(* IEC 61131-3 sources: axopen.templates/axopen.template.simple/ax/src/templates/unit, 7 files *)

(* ---- AutomatSequence.st ---- *)
NAMESPACE axosimple.UnitTemplate
    USING axosimple;
    USING AXOpen.Data;
    USING AXOpen.Core;
    USING System.Strings;

    ///<summary>
    /// Provides automatic mode sequence.
    ///</summary>
    {#ix-set:AttributeName = "<#AUTOMAT#>"}
    {S7.extern=ReadWrite}
    CLASS PUBLIC AutomatSequence
        EXTENDS AXOpen.Core.AxoSequencerContainer
        IMPLEMENTS IModeContainer
        VAR PUBLIC
            Steps : ARRAY[0..150] OF AXOpen.Core.AxoStep;
        END_VAR
        VAR PRIVATE
            Objs : axosimple.UnitTemplate.UnitObjects;
            _currentId : STRING;
        END_VAR

        METHOD INTERNAL Run
            VAR_INPUT
                inParent :  AXOpen.Core.IAxoObject;
                inUnitObjects : REF_TO axosimple.UnitTemplate.UnitObjects;
            END_VAR

            SUPER.Run(inParent);
        END_METHOD
        ///<summary>
        /// Contains logic of the steps of this sequence
        ///</summary>

        METHOD OVERRIDE Main
            // This sequecner executes the steps in cycles from top to bottom
            // in the same order they are written in the program
            // Each step in the sequence must can be used only once.
            // This sets the sequence to run in cycles (top-botton-top and again).
            THIS.SequenceMode := eAxoSequenceMode#Cyclic;

            IF (Steps[0].Execute(THIS, TRUE, '<#GET ID#>')) THEN
                //-------------------------------------------------------
                _currentId := 'newProducedPart';
                THIS.MoveNext();
                //-------------------------------------------------------
            END_IF;

            IF (Steps[10].Execute(THIS, TRUE, '<#GET DATA#>')) THEN
                //-------------------------------------------------------
                // IF(ProcessSettingsManager^.Read('MODEL_S').IsDone()) THEN
                //     ProcessDataManager^.DataManger.Payload := ProcessSettingsManager^.Payload;
                //     THIS.MoveNext();
                // END_IF;

                RETURN;

                IF (Objs.ProcessData.CreateOrUpdate(_currentId).IsDone()) THEN
                    THIS.MoveNext();
                END_IF;

                //-------------------------------------------------------
            END_IF;

            IF (Steps[20].Execute(THIS, TRUE, '<#DO SOMETHING#>')) THEN
                //-------------------------------------------------------

                IF(Objs.ProcessData.DataManger.Payload.JigDataMatrixCode.Inspect(THIS, '').Done()) THEN
                    THIS.MoveNext();
                END_IF;
                //-------------------------------------------------------
            END_IF;

            IF (Steps[30].Execute(THIS, TRUE, '<#DO SOMETHING#>')) THEN
                //-------------------------------------------------------
                IF(Objs.ProcessData.DataManger.Payload.PartPresence.Inspect(THIS, TRUE).Done()) THEN
                    THIS.MoveNext();
                END_IF;
                //-------------------------------------------------------
            END_IF;

            IF (Steps[4].Execute(THIS, TRUE, '<#DO SOMETHING#>')) THEN
                //-------------------------------------------------------
                IF(Objs.ProcessData.DataManger.Payload.RivetingPreasure.Inspect(THIS, 1.5).Done()) THEN
                    THIS.MoveNext();
                END_IF;
                //-------------------------------------------------------
            END_IF;

            IF (Steps[149].Execute(THIS, TRUE, '<#UPDATE DATA#>')) THEN
                //-------------------------------------------------------
                IF (Objs.ProcessData.Update(_currentId).IsDone()) THEN
                    THIS.MoveNext();
                END_IF;
                //-------------------------------------------------------
            END_IF;

            // This will close the sequence and will return to the first step.
            THIS.Close(Steps[150]);
        END_METHOD
    END_CLASS
END_NAMESPACE

(* ---- Components.st ---- *)
NAMESPACE axosimple.UnitTemplate
    USING axosimple;
    USING AXOpen.Data;
    USING AXOpen.Core;
    USING System.Strings;

    ///<summary>
    /// Groups components of this controller unit.
    ///</summary>
    {S7.extern=ReadWrite}
    CLASS Components
        EXTENDS AXOpen.Core.AxoObject
        VAR PUBLIC
            // HERE DECLARE COMPONENTS USED BY THIS CONTROLLED UNIT
            HorizontalCylinder : AXOpen.Components.Pneumatics.AxoCylinder;
            VerticalCylinder : AXOpen.Components.Pneumatics.AxoCylinder;
            GripperCylinder : AXOpen.Components.Pneumatics.AxoCylinder;
        END_VAR

        METHOD PUBLIC Update
            VAR_INPUT
                parent : IAxoObject;
                Inputs : ref_to axosimple.Inputs; // must be a ref_to due to arrays in components
                Outputs : ref_to axosimple.Outputs;
            END_VAR
            THIS.Initialize(parent);

            THIS.Initialize(parent);
            // HERE INITIALIZE YOUR COMPONENTS
            HorizontalCylinder.Run(THIS, Inputs^.P0[0], Inputs^.P0[1], Outputs^.P0[0], Outputs^.P0[1]);
            VerticalCylinder.Run(THIS, Inputs^.P0[2], Inputs^.P0[3], Outputs^.P0[2], Outputs^.P0[3]);
            GripperCylinder.Run(THIS, Inputs^.P0[4], Inputs^.P0[5], Outputs^.P0[4], Outputs^.P0[5]);

        END_METHOD
    END_CLASS
END_NAMESPACE

(* ---- GroundSequence.st ---- *)
NAMESPACE axosimple.UnitTemplate
    USING axosimple;
    USING AXOpen.Data;
    USING AXOpen.Core;
    USING System.Strings;

    ///<summary>
    /// Provides ground mode sequence.
    ///</summary>
    {#ix-set:AttributeName = "<#GROUND#>"}
    {S7.extern=ReadWrite}
    CLASS PUBLIC GroundSequence
        EXTENDS AXOpen.Core.AxoSequencerContainer
        IMPLEMENTS IModeContainer
        VAR PUBLIC
            Steps : ARRAY[0..20] OF AXOpen.Core.AxoStep;
            MoveToWork : AXOpen.Core.AxoTask;
        END_VAR
        VAR PRIVATE
            Objs : REF_TO axosimple.UnitTemplate.UnitObjects;
            Components : REF_TO axosimple.UnitTemplate.Components;

            ProcessDataManager : REF_TO axosimple.UnitTemplate.ProcessDataManager;
            ProcessSettingsManager : REF_TO axosimple.UnitTemplate.FragmentProcessDataManger;
            TechnologySettingsManager : REF_TO axosimple.UnitTemplate.TechnologyDataManager;

            PersistentSettingsManager : REF_TO AxoDataPersistentExchange;

            _currentId : STRING;

            techSetttingsId : STRING;
        END_VAR

        METHOD INTERNAL Run
            VAR_INPUT
                inParent : AXOpen.Core.IAxoObject;
                inUnitObjects : REF_TO axosimple.UnitTemplate.UnitObjects;
            END_VAR

            IF Objs = NULL THEN
                Objs := inUnitObjects;
            END_IF;

            SUPER.Run(inParent);

        END_METHOD
        ///<summary>
        /// Contains logic of the steps of this sequence
        ///</summary>

        METHOD PROTECTED OVERRIDE Main
            // IF (Components = NULL OR ProcessData = NULL) THEN
            //     RETURN;
            // END_IF;
            // This sequecner executes the steps in cycles from top to bottom
            // in the same order they are written in the program
            // Each step in the sequence must can be used only once.
            // This sets the sequence to run once (top-botton) and stops with done after closing.
            THIS.SequenceMode := eAxoSequenceMode#RunOnce;

            IF (Steps[0].Execute(THIS, TRUE, '<#RESTORE#>')) THEN
                //-------------------------------------------------------
                    TechnologySettingsManager^.Restore();
                    ProcessSettingsManager^.Restore();
                    ProcessDataManager^.Restore();

                    THIS.MoveNext();
                //-------------------------------------------------------
            END_IF;

            IF (Steps[1].Execute(THIS, TRUE, '<#READ PERSISTENT SETTINGS#>')) THEN
                //-------------------------------------------------------
                CASE TO_INT( THIS.GetMicroStepValue()) OF
                    0 :
                        IF PersistentSettingsManager^.InvokeRead(THIS,'UnitTemplate') THEN
                            THIS.SetMicroStepValue(UINT#10);
                        END_IF;
                    10 :
                        IF PersistentSettingsManager^.IsReadDone(THIS) THEN
                                THIS.MoveNext();
                        END_IF;
                    ELSE
                        THIS.SetMicroStepValue(UINT#0);
                END_CASE;
                //-------------------------------------------------------
            END_IF;

            IF (Steps[5].Execute(THIS, TRUE, '<#READ TECHNOLOGY SETTINS#>')) THEN
                //-------------------------------------------------------
                IF CurrentStep.IsFirstEntryToStep() THEN

                    IF Objs^.Global^.TechnologySettings^.Common.Entity.DataEntityId <> '' THEN
                       techSetttingsId := Objs^.Global^.TechnologySettings^.Common.Entity.DataEntityId; // TAKE GLOGAL TECHNOLOGY SETTINGS ID

                    ELSIF Objs^.TechnologySettings^.Payload.DataEntityId <> '' THEN // TAKE LAST LOADED FOR STATION
                        techSetttingsId := Objs^.TechnologySettings^.Payload.DataEntityId;

                    ELSIF Objs^.LastTechnologySettings <> '' THEN // TAKE LAST LOADED FROM PERSISTENT
                        techSetttingsId := Objs^.LastTechnologySettings;
                    ELSE
                        Objs^.LastTechnologySettings := 'default'; // FORCE DEFAULT VALUE
                        techSetttingsId := Objs^.LastTechnologySettings;
                    END_IF;

                    IF Objs^.Global^.TechnologySettings^.Common.Entity.DataEntityId = Objs^.TechnologySettings^.Payload.DataEntityId then
                        //THIS.MoveNext(); // you can skip loading...
                        ;
                    end_if;

                else
                    IF(TechnologySettingsManager^.Read( techSetttingsId ).IsDone()) THEN
                        THIS.MoveNext();
                    END_IF;
                END_IF;
                //-------------------------------------------------------
            END_IF;

            IF (Steps[3].Execute(THIS, TRUE, '<#DO SOMETHING#>')) THEN
                //-------------------------------------------------------
                IF CurrentStep.Duration > TIME#2s THEN
                    THIS.MoveNext();
                END_IF;
                //-------------------------------------------------------
            END_IF;

            IF (Steps[19].Execute(THIS, TRUE, '<#SAVE DATA#>')) THEN
                //-------------------------------------------------------
                CASE TO_INT( THIS.GetMicroStepValue()) OF
                    0 :
                        IF ProcessDataManager^.Shared.Entity.DataEntityId <> '' THEN
                            _currentId := ProcessDataManager^.Shared.Entity.DataEntityId;
                            THIS.SetMicroStepValue(UINT#10);

                        ELSE // FIST RUN OR WITHOUT DATA
                            THIS.MoveNext();
                        END_IF;

                    10 : // update part as a corrupted a interrupted
                        ProcessDataManager^.Shared.Entity.WasReset := true;
                        IF ProcessDataManager^.Update(_currentId).IsDone() THEN
                                THIS.MoveNext();
                        END_IF;
                    ELSE
                        THIS.SetMicroStepValue(UINT#0);
                END_CASE;
                //-------------------------------------------------------
            END_IF;

            // This will close the sequence and will return to the first step.
            THIS.Close(Steps[20]);
        END_METHOD
    END_CLASS
END_NAMESPACE

(* ---- ProcessData.st ---- *)
NAMESPACE axosimple.UnitTemplate
    USING axosimple;
    USING AXOpen.Data;
    USING AXOpen.Core;
    USING System.Strings;

    {S7.extern=ReadWrite}
    CLASS ProcessData
        EXTENDS AXOpen.Data.AxoDataEntity
        VAR PUBLIC
            Header : axosimple.UnitHeader;
            DimX    : AXOpen.Inspectors.AxoAnalogueInspector;
            DimY    : AXOpen.Inspectors.AxoAnalogueInspector;
            DimZ    : AXOpen.Inspectors.AxoAnalogueInspector;
        END_VAR
    END_CLASS
END_NAMESPACE

(* ---- ServiceMode.st ---- *)
NAMESPACE axosimple.UnitTemplate
    USING axosimple;
    USING AXOpen.Data;
    USING AXOpen.Core;
    USING System.Strings;

    ///<summary>
    /// Provides logic for service/manual/maintenance mode.
    ///</summary>
    {#ix-set:AttributeName = "<#SERVICE#>"}
    {S7.extern=ReadWrite}
    CLASS PUBLIC ServiceMode
        EXTENDS AXOpen.Core.AxoTask
        IMPLEMENTS IModeContainer
        ///<summary>
        /// Runs service mode logic. This method must be called cyclically.
        ///</summary>

        METHOD PUBLIC Run
            VAR_INPUT
                parent : AXOpen.Core.IAxoObject;
            END_VAR
            VAR_IN_OUT
                components : axosimple.UnitTemplate.Components;
            END_VAR
            THIS.Initialize(parent);
            IF THIS.Execute() THEN
                THIS.Handle(components);
            END_IF;
        END_METHOD

        METHOD PRIVATE Handle
            VAR_IN_OUT
                components : axosimple.UnitTemplate.Components;
            END_VAR
            ;
            // HERE CALL LOGIC FOR MANUAL/SERICE OPERATIONS

            components.DI_1.ActivateManualControl();
            components.DI_2.ActivateManualControl();
            // components.DI_3.ActivateManualControl();
            // components.DI_4.ActivateManualControl();

            components.DO_1.ActivateManualControl();
            components.DO_2.ActivateManualControl();
            // components.DO_3.ActivateManualControl();
            // components.DO_4.ActivateManualControl();

            components.AI_1.ActivateManualControl();
            components.AI_2.ActivateManualControl();
            // components.AI_3.ActivateManualControl();
            // components.AI_4.ActivateManualControl();

            components.AO_1.ActivateManualControl();
            components.AO_2.ActivateManualControl();
            // components.AO_3.ActivateManualControl();
            // components.AO_4.ActivateManualControl();

            components.Cylinder_1.ActivateManualControl();
            components.Cylinder_2.ActivateManualControl();
            // components.Cylinder_3.ActivateManualControl();
            // components.Cylinder_4.ActivateManualControl();

            // components.Reader_1.ActivateManualControl();
            // components.Reader_2.ActivateManualControl();

            // components.Camera_1.ActivateManualControl();
            // components.Camera_2.ActivateManualControl();

            // components.Drive_R1.ActivateManualControl();
            // components.Drive_R2.ActivateManualControl();

            // components.Drive_F1.ActivateManualControl();
            // components.Drive_F2.ActivateManualControl();

        END_METHOD
    END_CLASS
END_NAMESPACE

(* ---- Unit.st ---- *)
NAMESPACE axosimple.UnitTemplate
    USING axosimple;
    USING AXOpen.Data;
    USING AXOpen.Core;
    USING System.Strings;

    ///<summary>
    /// Represents controlled units and high level task coordination.
    ///</summary>
    {S7.extern=ReadWrite}
    CLASS Unit
        EXTENDS axosimple.BaseUnit.UnitBase
        VAR PUBLIC
            ///<summary>
            /// Provide access to unit objets, that are used into sequnces.
            ///</summary>
            UnitObjects  : axosimple.UnitTemplate.UnitObjects;

            ///<summary>
            /// Ground sequence. Contains logic that brings the unit into initial state.
            ///</summary>
            GroundSequence : axosimple.UnitTemplate.GroundSequence;

            ///<summary>
            /// Automatic sequence. Contains logic for automatic operations of this unit.
            ///</summary>
            AutomatSequence : axosimple.UnitTemplate.AutomatSequence;

            ///<summary>
            /// Service mode contains logic for service/manual operations.
            ///</summary>
            ServiceMode : axosimple.UnitTemplate.ServiceMode;
        END_VAR
        ///<summary>
        /// Runs this unit.
        ///</summary>

        METHOD PUBLIC Run
            VAR_INPUT
                parent : IAxoContext;
            END_VAR
            VAR_IN_OUT
                ///<summary>
                /// Hardware input structure
                ///</summary>
                Inputs : axosimple.Inputs;
                ///<summary>
                /// Hardware output structure
                ///</summary>
                Outputs : axosimple.Outputs;
            END_VAR
            VAR_INPUT
                TechnologySettings : REF_TO axosimple.UnitTemplate.FragmentTechnologyDataManger;
                ProcessSettings : REF_TO axosimple.UnitTemplate.FragmentProcessDataManger;
                Global : REF_TO axosimple.GlobalContextObjects;
            END_VAR
            THIS.Initialize(parent);
            UnitObjects.ProcessSettings := ProcessSettings;
            UnitObjects.TechnologySettings := TechnologySettings;
            UnitObjects.G := Global;
            THIS.Execute(Inputs, Outputs);
        END_METHOD

        METHOD PRIVATE Execute
            VAR_IN_OUT
                Inputs : axosimple.Inputs;
                Outputs : axosimple.Outputs;
            END_VAR

            // Component I/O immange and management handling.
            UnitObjects.Components.Update(THIS, Inputs, Outputs);
            // Process data manager
            UnitObjects.ProcessData.Run(THIS);
            // Process settings data manager
            UnitObjects.ProcessSettings^.Run(THIS);
            // Technology data manager
            UnitObjects.TechnologySettings^.Run(THIS);
            // Handles ground sequence
            GroundSequence.Run(THIS, REF(UnitObjects));

            // Restores other states when Ground executes
            IF (GroundSequence.IsBusy()) THEN
                AutomatSequence.Restore();
                ServiceMode.Restore();
            END_IF;

            // Handles automatic sequence (ground must be previously done)
            AutomatSequence.IsDisabled := GroundSequence.Status <> eAxoTaskState#Done;
            AutomatSequence.Run(THIS, REF(UnitObjects));
            // Handles service/manual mode
            ServiceMode.Run(THIS, UnitObjects.Components);

            IF ServiceMode.IsBusy() THEN
                GroundSequence.Restore();
                AutomatSequence.Restore();
            END_IF;

            // remember last selected technolgy identifier
            if  (UnitObjects.TechnologySettings^.Payload.DataEntityId <> '') THEN
                IF UnitObjects.LastTechnologySettings <> UnitObjects.TechnologySettings^.Payload.DataEntityId THEN
                    IF UnitObjects.G^.Persits^.InvokeUpdate(THIS, '') THEN
                        UnitObjects.LastTechnologySettings :=  UnitObjects.TechnologySettings^.Payload.DataEntityId;
                    END_IF;
                END_IF;
            END_IF;

        END_METHOD
    END_CLASS

END_NAMESPACE

(* ---- UnitObjects.st ---- *)
NAMESPACE axosimple.UnitTemplate

    USING axosimple;
    USING AXOpen.Data;
    USING AXOpen.Core;
    USING System.Strings;

    {S7.extern=ReadWrite}
    CLASS PUBLIC UnitObjects EXTENDS axosimple.BaseUnit.UnitObjects
        VAR PUBLIC
            ///<summary>
            /// Handles and intializes components used by this unit.
            ///</summary>
            C : axosimple.UnitTemplate.Components;

            ///<summary>
            /// Provides access to process data manager of this unit.
            ///</summary>
            PD : axosimple.UnitTemplate.ProcessDataManager;

            ///<summary>
            /// Provides access to technology data manager of this unit.
            ///</summary>
            TD : axosimple.UnitTemplate.TechnologyDataManager;

            // ///<summary>
            // /// Provides access to technology settings of this unit.
            // ///</summary>
            // TS : REF_TO axosimple.UnitTemplate.TechnologyDataExchange;

            // ///<summary>
            // /// Provides access to process setting of this unit.
            // ///</summary>
            // PS : REF_TO axosimple.UnitTemplate.ProcessDataExchange;

            {#ix-attr:[AXOpen.Data.PersistentAttribute("UnitTemplate")]}
            SpecialSettings :STRING[64] ;

            // https://ix-ax.github.io/AXOpen/core/docs/AXODIALOG.html#closing-a-dialog-with-external-signal
            _DL     : AXOpen.Core.AxoDialog;

            // https://ix-ax.github.io/AXOpen/core/docs/AXOALERTDIALOG.html#invoking-alerts-from-plc
            _ADL    : AXOpen.Core.AxoAlert;

            // it needs to be handle from auto or ground sequnce
            _IDL    : AXOpen.Inspectors.AxoInspectorDialog;

        END_VAR
    END_CLASS

END_NAMESPACE
